{attribute 'enable_dynamic_creation'}
FUNCTION_BLOCK FB_Slide EXTENDS FB_TargetBase
VAR_INPUT
END_VAR
VAR_OUTPUT
END_VAR
VAR
	
	//neue Slide Variablen
	stMarker1Position	: ST_3DPoint;
	stCamOffsetMarker1	: ST_3DPoint;
	stCamOffsetMarker2	: ST_3DPoint;
	rTargetRot			: REAL;			//Winkel * 1000	
END_VAR

METHOD FB_init : BOOL
VAR_INPUT
	bInitRetains : BOOL; // if TRUE, the retain variables are initialized (warm start / cold start)
	bInCopyCode : BOOL;  // if TRUE, the instance afterwards gets moved into the copy code (online change)
END_VAR
eObjectType := E_ObjectType.OBJECTTYPE_Slide;
eObjectGroup := E_ObjectGroup.OBJECTGROUP_Target;
END_METHOD

METHOD M_AddChild : ERRORID
VAR_INPUT
	pObject : POINTER TO FB_Object;
	nSlotNr	: UINT;
	nIndex 	: INT;
END_VAR
//Kann folgende Objekte aufnehmen:
IF pObject > 0 THEN
	IF pObject^.P_eObjectType = E_ObjectType.OBJECTTYPE_Point OR
		pObject^.P_eObjectType = E_ObjectType.OBJECTTYPE_Slide OR
		pObject^.P_eObjectType = E_ObjectType.OBJECTTYPE_Mtp OR
		(*pObject^.P_eObjectType = E_ObjectType.OBJECTTYPE_SpotPattern OR*)
		pObject^.P_eObjectType = E_ObjectType.OBJECTTYPE_SpotArray
		(*pObject^.P_eObjectType = E_ObjectType.OBJECTTYPE_TargetGroup OR
		pObject^.P_eObjectType = E_ObjectType.OBJECTTYPE_Wafer*) THEN
		M_AddChild := SUPER^.M_AddChild(pObject,nSlotNr,nIndex);
	ELSE
		M_AddChild := E_ErrorIdObjMgmt.ERRORID_InvalidParentObject;
	END_IF
ELSE
	M_AddChild := E_ErrorIdObjMgmt.ERRORID_InvalidParentObject;
END_IF
END_METHOD

METHOD M_Align : ST_3DPoint
VAR_INPUT
	stPos: ST_3DPoint;
END_VAR
VAR_OUTPUT
	lrAngle: LREAL;
END_VAR
VAR
	stPosTmp: ST_3DPoint;
END_VAR
//lrAngle := THIS^.lrAngle;
END_METHOD

METHOD M_CalcAngle : ERRORID
VAR_INPUT
END_VAR
(*IF bIsAligned THEN
	//Falls ein Fehler bei der Berechnung auftritt, wird "bIsAligned" zurückgesetzt
	lrAngle := F_GetTwoLineAngle(stMark1,stMark2,stMark1Act, stMark2Act);
	IF lrAngle = 9999.9 THEN
		bIsAligned := FALSE;
		lrAngle := 0.0;
	END_IF
ELSE
	lrAngle := 0.0;
END_IF*)
END_METHOD

METHOD M_ClearAllProps
VAR_INPUT
	bIgnoreParent : BOOL; //Es wird das gesamte OD gelöscht. -> Zeiger auf Parent nicht mehr gültig!
END_VAR
SUPER^.M_ClearAllProps(bIgnoreParent);
//bIsAligned:= FALSE;
END_METHOD

METHOD M_GetAbsPos : ST_3DPoint
VAR_INPUT
	pChildPos	: POINTER TO ST_3DPoint;
	eTargetRef 	: E_TargetRef;
	nParam1		: UINT;
 	nParam2		: UINT;
	nParam3		: USINT;
	nParam4		: USINT;
	nZLevel		: USINT;
END_VAR
VAR_OUTPUT
	nErrorId 	: ERRORID;
	lrAngle		: LREAL;

END_VAR
VAR
	stLocPos: ST_3DPoint;
	stLocPosAligned: ST_3DPoint;
	stNull: ST_3DPoint;
END_VAR
//Mit Alignment
IF NOT nParam4 > 0 THEN
	stLocPos := F_Add3DPoints(stRelPos,F_Add3DPoints(stLocPos,stCamOffsetMarker1));	//Cam Offset 1 von GUI übermittelt
	stLocPos.Z := stLocPos.Z + stDimension.Height + rZOffset;
	CASE eTargetRef OF
		E_TargetRef.TARGETREF_LeftBottom:		//Gcode M_SetStartZeroPoint nimmt immer TARGETREF_LeftBottom 
			;
		E_TargetRef.TARGETREF_LeftTop:
			stLocPos.Y := stLocPos.Y + stDimension.Depth ;
		E_TargetRef.TARGETREF_RightBottom:
			stLocPos.X := stLocPos.X + stDimension.Width;
		E_TargetRef.TARGETREF_RightTop:
			stLocPos.X := stLocPos.X + stDimension.Width;
			stLocPos.Y := stLocPos.Y + stDimension.Depth;
		E_TargetRef.TARGETREF_Center:
			stLocPos.X := stLocPos.X + stDimension.Width / 2.0;
			stLocPos.Y := stLocPos.Y + stDimension.Depth / 2.0;
		
	ELSE
		nErrorId := E_ErrorIdCmd.ERRORID_InvalidTargetPointRef;
	END_CASE
	
	IF nErrorId > 0 THEN
		RETURN;
	END_IF
	
	
	stLocPosAligned := stLocPos;
	
	IF rTargetRot <> 0 THEN	
		//Drehen
		stLocPosAligned := F_RotatePoint(stLocPosAligned,F_Add3DPoints(stMarker1Position,stCamOffsetMarker1),rTargetRot/1000);
	END_IF
	
	
	IF pChildPos > 0 THEN
			lrAngle := rTargetRot/1000;
		//IF THIS^.rTargetRot <> 0 THEN
			pChildPos^ := F_RotatePoint(pChildPos^,stNull,rTargetRot/1000);
			//END_IF
			pChildPos^.X := pChildPos^.X + stLocPosAligned.X -stLocPos.X;
			pChildPos^.Y := pChildPos^.Y + stLocPosAligned.Y -stLocPos.Y;
		
		stLocPos.X := pChildPos^.X + stLocPos.X;
		stLocPos.Y := pChildPos^.Y + stLocPos.Y;
		stLocPos.Z := pChildPos^.Z + stLocPos.Z;	
		
	ELSE
		stLocPos := stLocPosAligned;
	END_IF
	ELSE
	//Alignment ignorieren
	stLocPos := F_Sub3DPoints(stRelPos,stLocPos);	//Cam Offset 1 von GUI übermittelt
	stLocPos.Z := stLocPos.Z + stDimension.Height + rZOffset;
	CASE eTargetRef OF
		E_TargetRef.TARGETREF_LeftBottom:		//Gcode M_SetStartZeroPoint nimmt immer TARGETREF_LeftBottom 
			;
		E_TargetRef.TARGETREF_LeftTop:
			stLocPos.Y := stLocPos.Y + stDimension.Depth ;
		E_TargetRef.TARGETREF_RightBottom:
			stLocPos.X := stLocPos.X + stDimension.Width;
		E_TargetRef.TARGETREF_RightTop:
			stLocPos.X := stLocPos.X + stDimension.Width;
			stLocPos.Y := stLocPos.Y + stDimension.Depth;
		E_TargetRef.TARGETREF_Center:
			stLocPos.X := stLocPos.X + stDimension.Width / 2.0;
			stLocPos.Y := stLocPos.Y + stDimension.Depth / 2.0;
		
	ELSE
		nErrorId := E_ErrorIdCmd.ERRORID_InvalidTargetPointRef;
	END_CASE
	
	IF nErrorId > 0 THEN
		RETURN;
	END_IF
	
	
	stLocPosAligned := stLocPos;
	
	IF rTargetRot <> 0 THEN	
		//Drehen
		//stLocPosAligned := F_RotatePoint(stLocPosAligned,F_Add3DPoints(stMarker1Position,stCamOffsetMarker1),-rTargetRot/1000);
	END_IF
	
	
	IF pChildPos > 0 THEN
			lrAngle := rTargetRot/1000;
		//IF THIS^.rTargetRot <> 0 THEN
			//pChildPos^ := F_RotatePoint(pChildPos^,stNull,-rTargetRot/1000);
			//END_IF
			pChildPos^.X := pChildPos^.X + stLocPosAligned.X -stLocPos.X;
			pChildPos^.Y := pChildPos^.Y + stLocPosAligned.Y -stLocPos.Y;
		
		stLocPos.X := pChildPos^.X + stLocPos.X;
		stLocPos.Y := pChildPos^.Y + stLocPos.Y;
		stLocPos.Z := pChildPos^.Z + stLocPos.Z;	
		
	ELSE
		stLocPos := stLocPosAligned;
	END_IF
	
END_IF

IF pParentTarget > 0 THEN
	IF pParentSlot > 0 THEN
 		stLocPos := pParentTarget^.M_GetAbsPos(pChildPos := ADR(stLocPos), eTargetRef:= E_TargetRef.TARGETREF_Slot,
													nParam1:= pParentSlot^.P_nNr,
													nParam2:= 0, nParam3:= 0, nParam4:= nParam4 ,nZLevel:= 0,
													lrAngle => lrAngle, nErrorId=> nErrorId);
	ELSE
 		stLocPos := pParentTarget^.M_GetAbsPos(pChildPos := ADR(stLocPos), eTargetRef:= E_TargetRef.TARGETREF_LeftBottom,
													nParam1:= 0,
													nParam2:= 0, nParam3:= 0, nParam4:= nParam4, nZLevel:= 0,
													lrAngle => lrAngle, nErrorId=> nErrorId);
	END_IF
END_IF

IF nErrorId > 0 THEN
	RETURN;
END_IF


M_GetAbsPos := stLocPos;
END_METHOD

METHOD M_GetAllProps : ERRORID
VAR_INPUT
	refCmdData : REFERENCE TO ST_CmdData;
END_VAR
SUPER^.M_GetAllProps(refCmdData); //wurde auskommentiert weil die Specific Points ein Relikt aus einer alten Version sind und nicht mehr gebraucht werden

//Alignment-Marken
	nCurrentPropIndex := 1;
	nCurrentPropIndex := nCurrentPropIndex + 1;
	refCmdData.n32Data[nCurrentPropIndex] := REAL_TO_DINT(stRelPos.X);				//2
	nCurrentPropIndex := nCurrentPropIndex + 1;                         			
	refCmdData.n32Data[nCurrentPropIndex] := REAL_TO_DINT(stRelPos.Y);				//3
	nCurrentPropIndex := nCurrentPropIndex + 1;                         			
	refCmdData.n32Data[nCurrentPropIndex] := REAL_TO_DINT(stRelPos.Z);				//4		
	nCurrentPropIndex := nCurrentPropIndex + 1;                                 	
	refCmdData.n32Data[nCurrentPropIndex] := REAL_TO_DINT(stDimension.Width);		//5
	nCurrentPropIndex := nCurrentPropIndex + 1;                                 	
	refCmdData.n32Data[nCurrentPropIndex] := REAL_TO_DINT(stDimension.Depth);		//6
	nCurrentPropIndex := nCurrentPropIndex + 1;                                 	
	refCmdData.n32Data[nCurrentPropIndex] := REAL_TO_DINT(stDimension.Height);		//7
	nCurrentPropIndex := nCurrentPropIndex + 1;                                 	
	refCmdData.n32Data[nCurrentPropIndex] := REAL_TO_DINT(rZOffset);				//8
	nCurrentPropIndex := nCurrentPropIndex + 1;                                 	
	refCmdData.n32Data[nCurrentPropIndex] := REAL_TO_DINT(stMarker1Position.X );	//9
	nCurrentPropIndex := nCurrentPropIndex + 1;                                 	
	refCmdData.n32Data[nCurrentPropIndex] := REAL_TO_DINT(stMarker1Position.Y);		//10
	nCurrentPropIndex := nCurrentPropIndex + 1;
	refCmdData.n32Data[nCurrentPropIndex] := REAL_TO_DINT(stCamOffsetMarker1.X);	//11
	nCurrentPropIndex := nCurrentPropIndex + 1;
	refCmdData.n32Data[nCurrentPropIndex] := REAL_TO_DINT(stCamOffsetMarker1.Y);	//12
	nCurrentPropIndex := nCurrentPropIndex + 1;                                 
	refCmdData.n32Data[nCurrentPropIndex] := REAL_TO_DINT(stCamOffsetMarker1.Z);	//13
	nCurrentPropIndex := nCurrentPropIndex + 1;                                 
	refCmdData.n32Data[nCurrentPropIndex] := REAL_TO_DINT(rTargetRot);				//14
	nCurrentPropIndex := nCurrentPropIndex + 1;                                 
	refCmdData.n32Data[nCurrentPropIndex] := REAL_TO_DINT(stCamOffsetMarker2.X);	//15
END_METHOD

METHOD M_SetAllProps : ERRORID
VAR_INPUT
	refCmdData : REFERENCE TO  ST_CmdData;
END_VAR

VAR
	rTemp: REAL;
	bFlag: BOOL;
END_VAR
//Hier wird ausdrücklich nicht die Basisklasse aufgerufen, da nur hier gecheckt wird, ob sich die RelPos in XY und die Breite und
//Tiefe geändert haben um das Alignment zurückzusetzen.
nNoOfProps := 16;
//Relative Koordinaten
nCurrentPropIndex := 2;
rTemp := DINT_TO_REAL(refCmdData.n32Data[nCurrentPropIndex]);
IF rTemp <> stRelPos.X THEN
	stRelPos.X := rTemp;
	bFlag := TRUE;
END_IF
nCurrentPropIndex := nCurrentPropIndex + 1;	//3
rTemp := DINT_TO_REAL(refCmdData.n32Data[nCurrentPropIndex]);
IF rTemp <> stRelPos.Y THEN
	stRelPos.Y := rTemp;
	bFlag := TRUE;
END_IF
nCurrentPropIndex := nCurrentPropIndex + 1;	//4
rTemp := DINT_TO_REAL(refCmdData.n32Data[nCurrentPropIndex]);
IF rTemp <> stRelPos.Z THEN
	stRelPos.Z := rTemp;
	bFlag := TRUE;
END_IF

//Dimensionen
nCurrentPropIndex := nCurrentPropIndex + 1;	//5
rTemp := DINT_TO_REAL(refCmdData.n32Data[nCurrentPropIndex]);
IF rTemp <> stDimension.Width THEN
	stDimension.Width := rTemp;
	bFlag := TRUE;
END_IF
nCurrentPropIndex := nCurrentPropIndex + 1;	//6
rTemp := DINT_TO_REAL(refCmdData.n32Data[nCurrentPropIndex]);
IF rTemp <> stDimension.Depth THEN
	stDimension.Depth := rTemp;
	bFlag := TRUE;
END_IF
nCurrentPropIndex := nCurrentPropIndex + 1;	//7
rTemp := DINT_TO_REAL(refCmdData.n32Data[nCurrentPropIndex]);
IF rTemp <> stDimension.Height THEN
	stDimension.Height := rTemp;
	bFlag := TRUE;
END_IF
nCurrentPropIndex := nCurrentPropIndex + 1;	//8
rZOffset := DINT_TO_REAL(refCmdData.n32Data[nCurrentPropIndex]);

//Marker-Points
nCurrentPropIndex := nCurrentPropIndex + 1;	//9
rTemp := DINT_TO_REAL(refCmdData.n32Data[nCurrentPropIndex]);
IF rTemp <> stMarker1Position.X THEN
	stMarker1Position.X := rTemp;
	bFlag := TRUE;
END_IF

nCurrentPropIndex := nCurrentPropIndex + 1;	//10
rTemp := DINT_TO_REAL(refCmdData.n32Data[nCurrentPropIndex]);
IF rTemp <> stMarker1Position.Y THEN
	stMarker1Position.Y := rTemp;
	bFlag := TRUE;
END_IF

nCurrentPropIndex := nCurrentPropIndex + 1;	//11
rTemp := DINT_TO_REAL(refCmdData.n32Data[nCurrentPropIndex]);
IF rTemp <> stCamOffsetMarker1.X THEN
	stCamOffsetMarker1.X := rTemp;
	bFlag := TRUE;
END_IF

nCurrentPropIndex := nCurrentPropIndex + 1;	//12
rTemp := DINT_TO_REAL(refCmdData.n32Data[nCurrentPropIndex]);
IF rTemp <> stCamOffsetMarker1.Y THEN
	stCamOffsetMarker1.Y := rTemp;
	bFlag := TRUE;
END_IF

nCurrentPropIndex := nCurrentPropIndex + 1;	//13
rTemp := DINT_TO_REAL(refCmdData.n32Data[nCurrentPropIndex]);
IF rTemp <> stCamOffsetMarker1.Z THEN
	stCamOffsetMarker1.Z := rTemp;
	bFlag := TRUE;
END_IF

nCurrentPropIndex := nCurrentPropIndex + 1;	//14
rTemp := DINT_TO_REAL(refCmdData.n32Data[nCurrentPropIndex]);
IF rTemp <> rTargetRot THEN
	rTargetRot := rTemp;
	bFlag := TRUE;
END_IF

nCurrentPropIndex := nCurrentPropIndex + 1;	//15
rTemp := DINT_TO_REAL(refCmdData.n32Data[nCurrentPropIndex]);
IF rTemp <> stCamOffsetMarker2.X THEN
	stCamOffsetMarker2.X := rTemp;
	bFlag := TRUE;
END_IF

P_pWorkplate^.P_bCalcCollisHeight := TRUE;
END_METHOD

METHOD M_SetSingleProp : ERRORID
VAR_INPUT
	refCmdData: REFERENCE TO ST_CmdData;
END_VAR
VAR
	rTemp: REAL;
	bFlag: BOOL;
END_VAR
	//Hier wird die Basisklasse ausgelassen, da auf Änderung der RelPos und Dimensionen für das Rücksetzen des Alignments gecheckt wird.
	rTemp := DINT_TO_REAL(refCmdData.n32Data[0]);
	CASE refCmdData.aHeader[1] OF
		2:	//XPosRel
			IF rTemp <> stRelPos.X THEN
				stRelPos.X := rTemp;
				bFlag := TRUE; 	
			END_IF
		3:	//YPosRel
			IF rTemp <> stRelPos.Y THEN
				stRelPos.Y := rTemp;
				bFlag := TRUE; 	
			END_IF
		4:	//ZPosRel
			IF rTemp <> stRelPos.Z THEN
				stRelPos.Z := rTemp;
				bFlag := TRUE;
				P_pWorkplate^.P_bCalcCollisHeight := TRUE; 	
			END_IF
		5:	//Width
			IF rTemp <> stDimension.Width THEN
				stDimension.Width := rTemp;
				bFlag := TRUE;
			END_IF
		6:	//Depth
			IF rTemp <> stDimension.Depth THEN
				stDimension.Depth := rTemp;
				bFlag := TRUE;
			END_IF
		7:	//Height
			IF rTemp <> stDimension.Height THEN
				stDimension.Height := rTemp;
				bFlag := TRUE;
				P_pWorkplate^.P_bCalcCollisHeight := TRUE; 	
			END_IF
		8:	//ZOffset
			IF rTemp <> rZOffset THEN
				rZOffset := rTemp;
				bFlag := TRUE; 	
			END_IF
		9:	//Marker1Position.X
			IF rTemp <> stMarker1Position.X  THEN
				stMarker1Position.X  := rTemp;
				bFlag := TRUE; 	
			END_IF
		10:	//Marker1Position.Y
			IF rTemp <> stMarker1Position.Y THEN
				stMarker1Position.Y := rTemp;
				bFlag := TRUE; 	
			END_IF
		11:	//stCamOffsetMarker1.X
			IF rTemp <> stCamOffsetMarker1.X THEN
				stCamOffsetMarker1.X := rTemp;
				bFlag := TRUE; 	
			END_IF
		12:	//stCamOffsetMarker1.Y
			IF rTemp <> stCamOffsetMarker1.Y THEN
				stCamOffsetMarker1.Y := rTemp;
				bFlag := TRUE; 	
			END_IF		
		13:	//stCamOffsetMarker1.Z
			IF rTemp <> stCamOffsetMarker1.Z THEN
				stCamOffsetMarker1.Z := rTemp;
				bFlag := TRUE; 	
			END_IF
		14:	//rTargetRot
			 IF rTemp <> rTargetRot THEN
				rTargetRot := rTemp;
				bFlag := TRUE; 	
			END_IF
		15:	//stCamOffsetMarker2.X
			 IF rTemp <> stCamOffsetMarker2.X THEN
				stCamOffsetMarker2.X := rTemp;
				bFlag := TRUE; 	
			END_IF
	END_CASE
(*	IF bFlag AND bIsAligned THEN
		bIsAligned := FALSE;
		lrAngle := 0.0;
	END_IF	
ELSE
	IF (nSpecPropIndex + 1) = refCmdData.aHeader[1] THEN
		rZOffset := DINT_TO_REAL(refCmdData.n32Data[0]);
	ELSE
		M_SetSingleProp := SUPER^.M_SetSingleProp(refCmdData);
	END_IF	
END_IF*)
END_METHOD

PROPERTY P_lrAbsAngle : LREAL
GET
IF pParentTarget > 0 THEN
	P_lrAbsAngle := pParentTarget^.P_lrAbsAngle + rTargetRot/1000;
END_IF
END_GET
END_PROPERTY

PROPERTY P_lrAngle : LREAL
GET
P_lrAngle := rTargetRot/1000;
END_GET
SET
rTargetRot := P_lrAngle*1000;
END_SET
END_PROPERTY

PROPERTY P_rOffsetX : REAL
GET
(*IF bIsAligned THEN
	P_rOffsetX := stMark1Act.X - stMark1.X;
END_IF*)
END_GET
END_PROPERTY

PROPERTY P_rOffsetY : REAL
GET
(*IF bIsAligned THEN
	P_rOffsetY := stMark1Act.Y - stMark1.Y;
END_IF*)
END_GET
END_PROPERTY

PROPERTY P_stMark1 : ST_3DPoint
GET
//P_stMark1 := F_Add3DPoints(stMark1,P_stAbsPosLB);
END_GET
END_PROPERTY

END_FUNCTION_BLOCK

(* stored: Version 1.1.0.1, ProductVersion 3.1.4024.15
   POU FB_Slide: Id {5b7a5dd9-2b33-43ad-bcd7-0fe06e1b5747}, SpecialFunc None
   Method FB_init: Id {56fc60b8-f4b3-4c41-b98a-b802f5fdf311}
   Method M_AddChild: Id {b14ecd0a-f896-45de-b2d1-14af36895cbd}
   Method M_Align: Id {c40fc800-d5bf-4d61-bd1d-7a843145e0f0}
   Method M_CalcAngle: Id {f03a70ae-8de6-4cc4-9319-0c6f68098416}
   Method M_ClearAllProps: Id {c718db61-3307-4bd2-9d9d-fb5f6ed22660}
   Method M_GetAbsPos: Id {e41b5210-d059-4b46-944c-cecba9bb6d01}
   Method M_GetAllProps: Id {08a89092-e3d0-4922-a9e7-445ae2dd7d3c}
   Method M_SetAllProps: Id {dd18b387-7fad-4b62-ac69-af937d567be9}
   Method M_SetSingleProp: Id {c5c11bee-3814-4093-9c74-828f9241e9ae}
   Property P_lrAbsAngle: Id {fc6d8818-1f1e-4f74-b8ed-785bf728a881}
   Get Get: Id {aa8a689c-0410-40f4-acf9-750142bb78b0}
   Property P_lrAngle: Id {a68f91b2-ff26-4a97-9785-c4a79e07200d}
   Get Get: Id {c70936ba-73d3-4a69-b12e-9e5bfce347f1}
   Set Set: Id {4d3507b9-4903-4d65-9193-ab31d1a7be27}
   Property P_rOffsetX: Id {1fe7a835-31f8-42c7-a085-4e07fe2efb0e}
   Get Get: Id {1c603615-7fbf-4ad1-b6ed-911e1925acb8}
   Property P_rOffsetY: Id {fa7f0748-c6aa-4535-a70b-4c0d35e8484c}
   Get Get: Id {5fdaa1e3-958d-4285-9953-c629f5ba1108}
   Property P_stMark1: Id {314481a6-4a9b-49c9-9deb-1c39931a181c}
   Get Get: Id {6822c0bd-729a-4f75-9d59-2600da50857c} *)
